FUNCTION_BLOCK FB_ErrorHandler

VAR_INPUT
END_VAR

VAR_OUTPUT
	bErrorResolved : BOOL;
END_VAR

VAR
END_VAR

//bErrorResolved := (* Verdadeiro quando o erro for resolvido

END_FUNCTION_BLOCK

(* stored: Version 1.1.0.1, ProductVersion 3.1.4024.12
   POU FB_ErrorHandler: Id {ed3260d9-d359-4ae7-aa35-a2a28acdd00d}, SpecialFunc None *)
